{attribute 'linkalways'} 
{attribute 'no_explicit_call' := 'This FB is a CLASS and must be accessed using methods or properties'}
{attribute 'enable_dynamic_creation'}
FUNCTION_BLOCK Node_F_VN_FillContainer_TcVnVector4_DINT EXTENDS VisionNode
VAR
    ipContainer : _ITcVnContainer;
    aValue : _TcVnVector4_DINT;
    hrPrev : _HRESULT(S_OK);
    hresult : _HRESULT(S_OK);
END_VAR

METHOD PUBLIC  Clone : I_Node
VAR
    pNode : POINTER TO Node_F_VN_FillContainer_TcVnVector4_DINT;
END_VAR
pNode := __NEW(Node_F_VN_FillContainer_TcVnVector4_DINT);
Clone := pNode^;
END_METHOD

METHOD FB_init : BOOL
VAR_INPUT
    bInitRetains : BOOL; // if TRUE, the retain variables are initialized (warm start / cold start)
    bInCopyCode : BOOL;  // if TRUE, the instance afterwards gets moved into the copy code (online change)
END_VAR
AddInput('ipContainer', ipContainer);
AddInput('aValue', aValue);
AddInput('hrPrev', hrPrev);
AddOutput('ipContainer', ipContainer);
AddOutput('hresult',hresult);
END_METHOD

METHOD PROTECTED OnExecute
hresult.Value := F_VN_FillContainer_TcVnVector4_DINT(
    ipContainer := ipContainer.Value,
    aValue := aValue.Value,
    hrPrev:= hrPrev.Value);
END_METHOD

METHOD PUBLIC PreExecutionCheck
VAR_INPUT
    Check : I_PreExecutionChecks;
END_VAR
Check.IsTrue(ipContainer.IsValid, 'ipContainer must be a valid container');
Check.IsTrue(ipContainer.IsType(TC_GLOBAL_CONST_LIST.ContainerType_Vector_TcVnVector4_DINT), 'ipContainer contains incorrect type');
END_METHOD

END_FUNCTION_BLOCK

(* stored: Version 1.1.0.1, ProductVersion 3.1.4026.13
   POU Node_F_VN_FillContainer_TcVnVector4_DINT: Id {b7a724f3-f762-4a44-9c03-15c8576264d7}, SpecialFunc None
   Folder Constructor: Id {1e012353-f58e-4ffb-9181-1bab96b68276}
   Method Clone: Id {5b7cfc57-c91a-4b76-9b94-e7d49b64f309}
   Method FB_init: Id {a0a975ba-fcdc-4f6c-8fc4-8b4c753979bb}
   Method OnExecute: Id {a859497e-a90b-47ec-82a7-65fb6707a3c4}
   Method PreExecutionCheck: Id {c8a27638-93c8-414b-a9bf-ab41d65d1af4} *)
